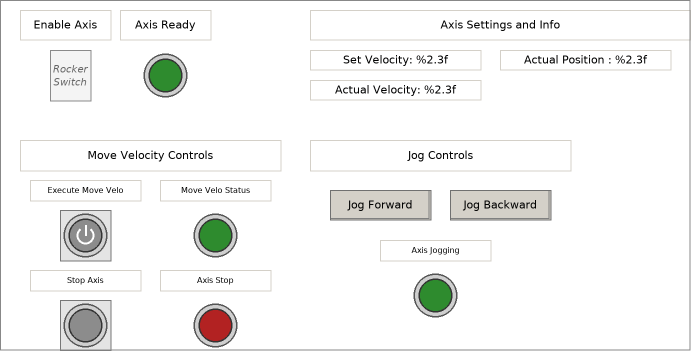
VISUALIZATION Visualization  // 691x351
    RockerSwitch (50,50 41x51), variable: MAIN.bEnable[1], behaviour: TOGGLE, style: Switch-RockerSwitch-Gray
    Lamp1 (140,50 51x51), variable: MAIN.bAxisReady[1], style: Lamp-Lamp1-Green
    Textfield (20,10 91x30), "Enable Axis"
    Textfield (120,10 91x30), "Axis Ready"
    Textfield (20,140 261x31), "Move Velocity Controls"
    PowerSwitch (60,210 51x51), variable: MAIN.bExeVelo[1], behaviour: TOGGLE, style: Switch-PowerSwitch-Gray
    Textfield (30,180 111x21), "Execute Move Velo"
    Textfield (310,10 381x30), "Axis Settings and Info"
    Textfield (500,50 171x20), "Actual Position : %2.3f", text variable: MAIN.ASI_Axis[1].Status.ActVelo
    Textfield (310,80 171x20), "Actual Velocity: %2.3f", text variable: MAIN.ASI_Axis[1].Status.ActVelo
    Textfield (310,50 171x20), "Set Velocity: %2.3f", text variable: MAIN.fSetVelo
        OnMouseUp: write the text variable via VisuDialogs.Numpad, min -500, max 2000
    Lamp1 (190,210 51x51), variable: MAIN.fbMoveVelo[1].Busy, style: Lamp-Lamp1-Green
    Textfield (160,180 111x21), "Move Velo Status"
    PushSwitch (60,300 51x51), variable: MAIN.bStop[1], behaviour: TOGGLE, style: Switch-PushSwitch-Gray
    Textfield (30,270 111x21), "Stop Axis"
    Textfield (160,270 111x21), "Axis Stop"
    Lamp1 (190,300 51x51), variable: MAIN.fbStop[1].Busy, style: Lamp-Lamp1-Red
    Textfield (310,140 261x31), "Jog Controls"
    Button (330,190 101x30), "Jog Forward"
        tap MAIN.bJogFwd[1]
    Button (450,190 101x30), "Jog Backward"
        tap MAIN.bJogBack[1]
    Lamp1 (410,270 51x51), variable: MAIN.fbJog[1].Busy, style: Lamp-Lamp1-Green
    Textfield (380,240 111x21), "Axis Jogging"
END_VISUALIZATION

(* stored: Version 1.1.0.1
   Visu Visualization: Id {a9ad9ddb-724f-4a3f-a5a5-ce490db95414} *)
